Fanuc KAREL source: kt00331.KL

-- PROVISIONAL review KL for V940-1; original PC SHA256 c0a76dd0d6f992c17e047a8a0152d5546236b22e87381a480792ecd43f614fde
-- Incomplete behavior may be omitted. Consult companion uncertainty JSON. Do not deploy.
PROGRAM KT00331
%NOLOCKGROUP
VAR
  I1 : INTEGER
  OUT : BOOLEAN
-- UNRESOLVED_DECL Y2 type=002018
BEGIN
  -- V9_ZERO_TABLE_METADATA_HINT layout=0001; no indexed target words; source/name/runtime held
  -- UNRESOLVED_PC offsets 5-16; opcodes 2E,23
  -- UNRESOLVED_PC offsets 21-35; opcodes 2E,22,9D,33,B2
  -- UNRESOLVED_PC offsets 40-62; opcodes 21,22,9D,33,B1,59,23
  -- UNRESOLVED_PC offsets 67-71; opcodes 7F
END KT00331
